INTERFACE iObjective

METHOD RegisterMover : BOOL
VAR_INPUT	
	NewMover		: REFERENCE TO Mover;
END_VAR
END_METHOD

METHOD UnregisterMover : BOOL
VAR_INPUT
	RemovingMover		: REFERENCE TO Mover;
END_VAR
END_METHOD

END_INTERFACE

(* stored: Version 1.1.0.1, ProductVersion 3.1.4024.9
   Itf iObjective: Id {1b7e0e94-0d7d-454a-b0fc-15c1ad212dac}
   Method RegisterMover: Id {1216fa06-f0b7-49bc-92d6-c03a5fb2af02}
   Method UnregisterMover: Id {32af6fa8-80c5-465d-bf8a-a0a9598a01a1} *)
